TYPE stXTSCfg :
STRUCT
	bInvertPolarity		: BOOL;
	udiNumStations		: UDINT;
	stStationsCfg 		: ARRAY [1..Tc3_XTS_Utility.TcIoXtsEnvironmentParameterList.MaxXtsInfoStation] OF stStationCfg;
END_STRUCT
END_TYPE

(* stored: Version 1.1.0.1, ProductVersion 3.1.4024.11
   DUT stXTSCfg: Id {d4f3e01a-17b4-4001-bf5c-b2d86a01486c} *)
